{attribute 'enable_dynamic_creation'}	
{attribute 'no_explicit_call' := 'do not call this function block directly'} 
FUNCTION_BLOCK FileOpenTask EXTENDS FileContentTask
VAR
	_ClassName : STRING := __POUNAME();

	_Open : Tc2_System.FB_FileOpen;
	_OpenMode : FILE_OPEN_MODE;
	_ContentHandlingMode : FILE_CONTENT_HANDLING_MODE;		
END_VAR

{attribute 'monitoring' := 'call'}
{attribute 'OPC.UA.DA.Property' := '1'}
PROPERTY AmsNetId : Tc2_System.T_AmsNetID
GET
AmsNetId := _Open.sNetId;
END_GET
SET
_Open.sNetId := AmsNetId;
END_SET
END_PROPERTY

{attribute 'monitoring' := 'call'}
PROPERTY ClassName : STRING
GET
ClassName := _ClassName;
END_GET
END_PROPERTY

{attribute 'monitoring' := 'call'}
{attribute 'OPC.UA.DA.Property' := '1'}
PROPERTY ContentHandlingMode : FILE_CONTENT_HANDLING_MODE
GET
ContentHandlingMode := _ContentHandlingMode;
END_GET
SET
_ContentHandlingMode := ContentHandlingMode;
END_SET
END_PROPERTY

METHOD Execute : BOOL
VAR_INPUT
	start : BOOL;
END_VAR
VAR
	
END_VAR
IF start THEN
	Validate();
	
	_Open(
		bExecute := FALSE,
		nMode := TO_DWORD(openMode) OR TO_DWORD(contentHandlingMode),
		tTimeout := Timeout 
	);	
END_IF

_Open(bExecute := TRUE);

IF _Open.bError THEN
	//exceptionFactory.ThrowException(__POSITION(), WStringHelper.Concat2("File open failed", GetErrorMessageByErrorId(_Open.nErrId)), __POUNAME(), ClassName, CurrentNamespace.Name, __POSITION(), _Open.nErrId);	
ELSIF NOT _Open.bBusy THEN
	FileContentManager.FilePath := _Open.sPathName;
	FileContentManager.OpenMode := _OpenMode;
	FileContentManager.ContentHandlingMode := _ContentHandlingMode;
	FileContentManager.PathType := _Open.ePath;
	FileContentManager.AmsNetId := _Open.sNetId;
	FileContentManager.FileHandle := _Open.hFile;
	
	Execute := EXECUTION_STATE.DONE;
END_IF
END_METHOD

{attribute 'monitoring' := 'call'}
{attribute 'OPC.UA.DA.Property' := '1'}
PROPERTY FilePath : Tc2_System.T_MaxString
GET
FilePath := _Open.sPathName;
END_GET
SET
_Open.sPathName := FilePath;
END_SET
END_PROPERTY

{attribute 'monitoring' := 'call'}
{attribute 'OPC.UA.DA.Property' := '1'}
PROPERTY OpenMode : FILE_OPEN_MODE
GET
OpenMode := _OpenMode;
END_GET
SET
_OpenMode := OpenMode;
END_SET
END_PROPERTY

{attribute 'monitoring' := 'call'}
{attribute 'OPC.UA.DA.Property' := '1'}
{attribute 'OPC.UA.DA.Access' := '1'}
PROPERTY PathType : E_OpenPath
GET
PathType := _Open.ePath;
END_GET
SET
_Open.ePath := PathType;
END_SET
END_PROPERTY

METHOD PROTECTED Validate
IF NOT __ISVALIDREF(FileContentManager) THEN
	//exceptionFactory.ThrowException(__POSITION(), "File content menager is not specified");
END_IF

IF FilePath = '' THEN
	//exceptionFactory.ThrowException(__POSITION(), "File path is not specified");
END_IF
END_METHOD

END_FUNCTION_BLOCK

(* stored: Version 1.1.0.1
   POU FileOpenTask: Id {cdd5f7ef-d507-46f5-a517-2d10f136b53b}, SpecialFunc None
   Property AmsNetId: Id {e0810aea-f2fb-48a8-903c-df260ce3d2d3}
   Get Get: Id {4897b848-77e1-4394-85d3-716e8e0cc1d9}
   Set Set: Id {fed7b16f-ac3a-45ec-a3bb-2e87753cea2e}
   Property ClassName: Id {089cfd8b-a488-4c5b-80c3-31bd17af5a4b}
   Get Get: Id {e5e61757-7352-4607-93e5-5695d606b197}
   Property ContentHandlingMode: Id {ba9bdbc6-6340-4d5f-bf60-84028fd6c118}
   Get Get: Id {2739e209-8bf2-4542-9cfd-a5408214b831}
   Set Set: Id {905cf5b8-a5d6-426c-a3d2-41a89f609b49}
   Method Execute: Id {ecadf39e-b907-480d-a969-8da6c5b792f2}
   Property FilePath: Id {d11eaf17-bdc4-431a-8d42-67a4a2039e6c}
   Get Get: Id {dc5d9aeb-64d4-4f09-9dd7-6d23a194f7e0}
   Set Set: Id {cda62e49-c241-4f3b-9fcc-bcbd7aba61df}
   Property OpenMode: Id {417d9a01-e4f3-41c3-b9ae-d701f1b0a94f}
   Get Get: Id {b6f938cd-0732-46fc-a01b-d17ad082814d}
   Set Set: Id {15090a11-58be-4c35-8b23-587d5b168d5e}
   Property PathType: Id {4e62d136-3c37-4e89-9a83-66775627a12a}
   Get Get: Id {91b7c649-fd0f-4567-8d7a-d2b7f2516f6e}
   Set Set: Id {72587730-2d56-446f-b736-71fe2489c287}
   Method Validate: Id {7f6e4b6c-5c82-44f6-b880-17a6bc43baf2} *)
